(* CODESYS project ABB-Codesys

Project tree, tasks and I/O mapping:
  PLC_AC500_V3 : PM5072-T-2ETH, ABB AG, order no. 1SAP124x00R0x73, version 3.8.1.0
    application Application
      task Task (cyclic, interval t#10ms, priority 14, watchdog t#20ms x 1) calls PLC_PRG
      Cam_2
      Cam
      CheckConfigurationObject
      program PLC_PRG [ST]
    Interfaces : Interfaces, ABB AG, version 3.8.1.0
      Ethernet : Ethernet, ABB AG, version 3.8.1.0
        ETH1 : Configuración de IP, ABB AG, version 3.8.1.0
          NetConfig : Configuración de red, ABB AG, version 3.8.0.0
        ETH2 : Configuración de IP, ABB AG, version 3.8.1.0
          NetConfig_1 : Configuración de red, ABB AG, version 3.8.0.0
        Protocols : Protocolos cliente, ABB AG, version 3.8.1.0
      OptionSlot_1
      OptionSlot_2
      OptionSlot_3
    IO_Bus : Bus de E/S, ABB AG, version 3.8.0.0
    OnBoard_IO : 12DI/8DO-T/2DC, ABB AG, version 3.8.1.0
        unmapped channels: Fast inputs DI0-DI3, Fast inputs DI4-DI7, Standard inputs DI8-DI11, Digital inputs - Transistor, Fast outputs DO0-DO3, Fast outputs DO4-DO7, Digital outputs - Transistor
    OnBoard_RTC : OnBoard RTC, ABB AG, version 3.8.0.0
*)

// PLC_AC500_V3/Application/PLC_PRG
PROGRAM PLC_PRG
VAR
	
	bool_1		:	BOOL;
	int_1		:	INT;
	FP_bool_1			:	Standard.R_TRIG;

END_VAR

FP_bool_1(CLK:=bool_1);

IF FP_bool_1.Q THEN
	int_1 := int_1 + 1;
END_IF

END_PROGRAM
